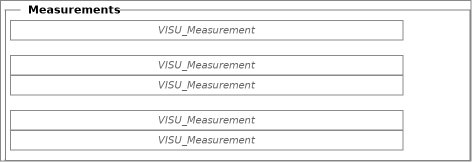
VISUALIZATION VISU_HydraulicsMeasurements  // 472x162
VAR_IN_OUT
	ref : Hydraulics;
    widget : HydraulicsWidget;
END_VAR
    Label (25,0 95x20), "Measurements"
    Frame (10,20 393x20)
        shows VISU_Measurement(widget := widget.bearingTemperature)
    Frame (10,55 393x20)
        shows VISU_Measurement(widget := widget.topFrequencyMeasurement)
    Frame (10,75 393x20)
        shows VISU_Measurement(widget := widget.topPressureMeasurement)
    Frame (10,110 393x20)
        shows VISU_Measurement(widget := widget.bottomFrequencyMeasurement)
    Frame (10,130 393x20)
        shows VISU_Measurement(widget := widget.bottomPressureMeasurement)
    Polyline (20,10) (5,10) (5,160) (470,160) (470,10) (120,10)
END_VISUALIZATION

(* stored: Version 1.1.0.1, ProductVersion 3.1.4019.2
   Visu VISU_HydraulicsMeasurements: Id {82d6451f-df1a-4cef-ad54-23365b06b00b} *)
